Universal Robots PolyScope program: annaetest.urp

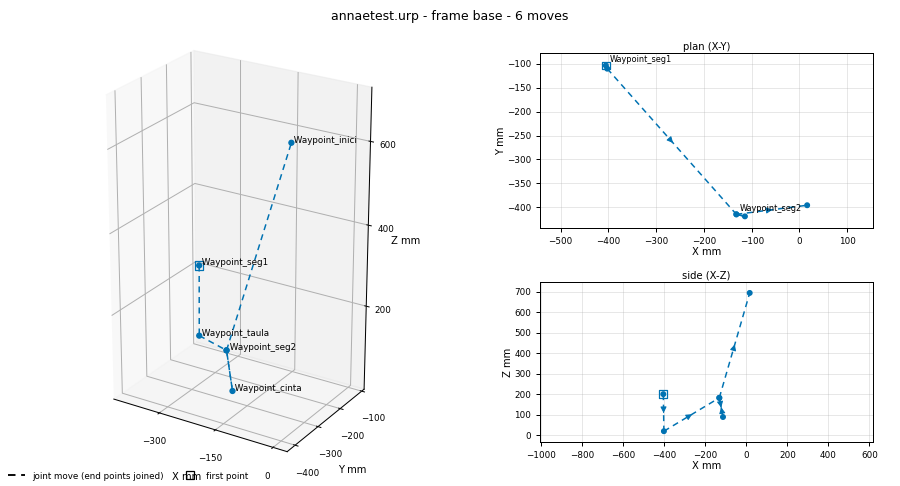
[picture p0: tool path of annaetest.urp in frame base, 6 of 6 moves have a stored position in this frame; points joined in program order, loops and branches not executed]
Program annaetest (installation=default directory=/programs createdIn=5.14.5 lastSavedIn=5.14.5 robotSerialNumber=20195300809)
Calibrated DH parameters: a=[-0.000085, -0.20076, -0.212369, 0.000121, -0.000118, 0]; d=[0.15185, -26.306375, 24.753047, 1.684739, 0.085386, 0.092088]; alpha=[1.572149, -0.00522, -0.011864, 1.571339, -1.571085, 0]; deltaTheta=[0, 0.599885, -0.513355, -0.086555, 0.000006, 0]
InitVariablesNode
BeforeStart
  SafeHome (positionOptionType=SPEED_AND_ACCELERATION speed=1.047198 acceleration=1.396263 nextMotionTime=2)
  URCap Gripper Activate (Robotiq_Grippers, Robotiq Inc.) dataModel(ResetAndActivateKey=false)
  URCap Gripper (Robotiq_Grippers, Robotiq Inc.) dataModel(position=0.0, force=0.0, speed=0.0, positionInDouble=0.0, forceInDouble=0.0, speedInDouble=0.0, slaveIds=[9], blocking=true)
  Set DigitalOutput pin=digital_out[0]; digitalValue=0
Robot Program (runOnlyOnce=false)
  MoveJ speed 60 deg/s, acceleration 80 deg/s^2 (useActiveTCP=true) feature=Base
    Waypoint Waypoint_seg1: TCP in base x=-405.501 y=-103.329 z=200.539 mm, rx=-0.0048 ry=3.1269 rz=0.0184 rad; joints [-3.586, -55.811, 23.808, -57.208, -91.526, -93.361] deg; TCP offset x=0 y=0 z=174 mm, rx=0 ry=0 rz=0 rad
  MoveJ speed 60 deg/s, acceleration 80 deg/s^2 (useActiveTCP=true) feature=Base
    Waypoint Waypoint_taula: TCP in base x=-402.597 y=-109.929 z=19.782 mm, rx=-0.0063 ry=3.107 rz=0.0042 rad; joints [-2.961, -60.266, 81.201, -108.983, -91.069, -93.359] deg
    Wait Sleep waitTime=3
    URCap Gripper (Robotiq_Grippers, Robotiq Inc.) dataModel(position=100.0, force=0.0, speed=0.0, positionInDouble=100.0, forceInDouble=0.0, speedInDouble=0.0, slaveIds=[9], blocking=true)
    MoveJ speed 60 deg/s, acceleration 80 deg/s^2 (useActiveTCP=true) feature=Base
      Waypoint Waypoint_seg2: TCP in base x=-132.21 y=-414.919 z=182.563 mm, rx=0.0272 ry=3.0978 rz=-0.0233 rad; joints [53.082, -54.709, 27.545, -62.075, -88.307, -35.588] deg
      Wait Sleep waitTime=2
      Waypoint Waypoint_cinta: TCP in base x=-114.289 y=-419.149 z=89.049 mm, rx=-0.0151 ry=3.1292 rz=-0.0074 rad; joints [56.598, -61.67, 65.025, -93.205, -90.122, -33.948] deg
      URCap Gripper (Robotiq_Grippers, Robotiq Inc.) dataModel(position=0.0, force=0.0, speed=0.0, positionInDouble=0.0, forceInDouble=0.0, speedInDouble=0.0, slaveIds=[9], blocking=true)
      Wait Sleep waitTime=2
      Waypoint Waypoint_seg2: TCP in base x=-132.21 y=-414.919 z=182.563 mm, rx=0.0272 ry=3.0978 rz=-0.0233 rad; joints [53.082, -54.709, 27.545, -62.075, -88.307, -35.588] deg
      Waypoint Waypoint_inici: TCP in base x=16.046 y=-395.898 z=694.328 mm, rx=-0.1219 ry=2.1863 rz=-2.2108 rad; joints [-1.741, -85.882, -10.156, -79.017, 5.245, -6.893] deg
      Set DigitalOutput pin=digital_out[0]; digitalValue=1
      Wait Sleep waitTime=2
      Set DigitalOutput pin=digital_out[0]; digitalValue=0
